{attribute 'GeneratedUsingTerminal: EK1122-0000-0018'}
{attribute addProperty BoxType "EK1122-0000-0018"}
{attribute addProperty Id "Beckhoff_ATH2xxxsub_EK1100EK1100_AB5A94672A_0001_ATH2000_0250_0022A_0001_ATH2000_0250_0022_83BFFE5D14A_0002_ATH2000_0250_0023A_0002_ATH2000_0250_0023_C3C2AA1314A_0003_ATH2000_0250_0024ATH2000_86175B4184A_0004_ATH2040_0250_0022ATH2040_86175B4184A_0005_ATH2040_0250_0023ATH2040_86175B4184A_0006_ATH2040_0250_0024ATH2040_86175B4184A_0007_ATH2050_0500_0022ATH2050_86175B4184A_0008_ATH2050_0500_0023ATH2050_86175B4184A_0009_ATH2050_0500_0024ATH2050_86175B4184A_0010_ATH2050_0501_0022ATH2050_86175B4184A_0011_ATH2050_0501_0023ATH2050_86175B4184A_0012_ATH2050_0501_0024ATH2050_86175B4184"}
{attribute addProperty CRC "2333965052"}
{attribute addProperty Size "870"}
TYPE Beckhoff_ATH2xxxEK1122_8B1D7AFC EXTENDS EK1122_AB5A9467 :
STRUCT
	{attribute addProperty Name "Beckhoff_ATH2xxxsub_EK1100"}
	Beckhoff_ATH2xxxsub_EK1100 : EK1100_AB5A9467;
	{attribute addProperty Name "A_0001_ATH2000_0250_0022"}
	A_0001_ATH2000_0250_0022 : A_0001_ATH2000_0250_0022_83BFFE5D;
	{attribute addProperty Name "A_0002_ATH2000_0250_0023"}
	A_0002_ATH2000_0250_0023 : A_0002_ATH2000_0250_0023_C3C2AA13;
	{attribute addProperty Name "A_0003_ATH2000_0250_0024"}
	A_0003_ATH2000_0250_0024 : ATH2000_86175B41;
	{attribute addProperty Name "A_0004_ATH2040_0250_0022"}
	A_0004_ATH2040_0250_0022 : ATH2040_86175B41;
	{attribute addProperty Name "A_0005_ATH2040_0250_0023"}
	A_0005_ATH2040_0250_0023 : ATH2040_86175B41;
	{attribute addProperty Name "A_0006_ATH2040_0250_0024"}
	A_0006_ATH2040_0250_0024 : ATH2040_86175B41;
	{attribute addProperty Name "A_0007_ATH2050_0500_0022"}
	A_0007_ATH2050_0500_0022 : ATH2050_86175B41;
	{attribute addProperty Name "A_0008_ATH2050_0500_0023"}
	A_0008_ATH2050_0500_0023 : ATH2050_86175B41;
	{attribute addProperty Name "A_0009_ATH2050_0500_0024"}
	A_0009_ATH2050_0500_0024 : ATH2050_86175B41;
	{attribute addProperty Name "A_0010_ATH2050_0501_0022"}
	A_0010_ATH2050_0501_0022 : ATH2050_86175B41;
	{attribute addProperty Name "A_0011_ATH2050_0501_0023"}
	A_0011_ATH2050_0501_0023 : ATH2050_86175B41;
	{attribute addProperty Name "A_0012_ATH2050_0501_0024"}
	A_0012_ATH2050_0501_0024 : ATH2050_86175B41;
END_STRUCT
END_TYPE

(* stored: Version 1.2.0.0, ProductVersion 3.1.4024.9
   DUT Beckhoff_ATH2xxxEK1122_8B1D7AFC: Id {4b4bd1ab-55d0-4e3b-9a04-bdadb43c8496} *)
